FUNCTION_BLOCK FB_MSSQL_spGetPartHistory
VAR_INPUT
	Execute					: BOOL;
	Enable					: BOOL;
	Reset					: BOOL;
END_VAR
VAR_OUTPUT
	Error					: BOOL;
	ErrorID					: DINT;
	Done					: BOOL;
	Busy					: BOOL;
	tcMessage 				: I_TcMessage;
	Q_tElapsedTime			: TIME;
	Result					: STRING(DB.MAX_STRING_SIZE);
END_VAR
VAR
	RTRIG_Execute			: R_TRIG;
	RTRIG_Reset				: R_TRIG;
	iState					: INT := -1;
	TON_Read				: TON;
	return_value	: DINT;
END_VAR
VAR_IN_OUT
	fbSQLResult				: FB_SQLResultEvt;
	fbSQLStoredProcedure	: FB_SQLStoredProcedureEvt;
END_VAR

RTRIG_Reset(CLK := Reset);
IF RTRIG_Reset.Q AND Execute AND Error AND NOT Busy THEN
	Execute := FALSE;
END_IF

RTRIG_Execute(CLK := Execute AND Enable);
IF(RTRIG_Execute.Q) THEN
	 Done							:= FALSE;
	 Error							:= FALSE;
	 ErrorID						:= 0;
	 
	 iState							:= 0;
ELSIF NOT Execute AND NOT Busy THEN
	Busy			:= FALSE;
	Done			:= FALSE;
	Error			:= FALSE;
	
	iState := -1;
END_IF
 
 // Elapsed Time
 TON_Read(PT:= T#5S);
 
 CASE iState OF
 
	 0:
	 		TON_Read.IN 						:= FALSE;
			Busy								:= TRUE;
			iState 								:= 10;
		
	10:
		IF fbSQLStoredProcedure.ExecuteDataReturn(pParameterStrc := 0, cbParameterStrc:= 0, pSQLDBResult := ADR(fbSqlResult)) THEN
			TON_Read.IN := TRUE;
			IF fbSQLStoredProcedure.bError THEN
				tcMessage := fbSQLStoredProcedure.ipTcResult;
				
				iState 							:= 1010;
			ELSE
				iState 							:= 20;
			END_IF    
		END_IF
		
	20:
		IF fbSQLResult.Read(0, fbSQLResult.nDataCount, ADR(Result), SIZEOF(Result), FALSE, TRUE) THEN
			IF fbSQLResult.bError THEN
				iState 							:= 1020;
			ELSE
				
				iState 							:= 30;
			END_IF
		END_IF
		
	30: 
		IF fbSQLResult.Release() THEN
			iState 								:= 999;	
		END_IF
		
	999:
		TON_Read.IN 	:= FALSE;
		Done			:= TRUE;
		Busy			:= FALSE;
		
 END_CASE 
 
IF iState > 1000 THEN
	Error 		:= TRUE;
	ErrorID	 	:= iState;
	Busy	 	:= FALSE;
	TON_Read.IN := FALSE;
	iState := -1;
END_IF

END_FUNCTION_BLOCK

(* stored: Version 1.1.0.1, ProductVersion 3.1.4024.15
   POU FB_MSSQL_spGetPartHistory: Id {9190f0a5-71ba-4c3a-9414-d2bb3a1b834a}, SpecialFunc None *)
